// TIA Portal V20 export
// export: Created 2026-04-20T18:50:18.1743947Z, ExportSetting WithDefaults, DisplayName Totally Integrated Automation Portal, DisplayVersion V20, DisplayName TIA Portal Openness, DisplayVersion V20, DisplayName TIA Portal Version Control Interface, DisplayVersion V20, DisplayName STEP 7 Professional, DisplayVersion V20, DisplayName STEP 7 Safety, DisplayVersion V20, DisplayName WinCC Basic/Comfort/Advanced, DisplayVersion V20
TYPE "UDT_AlarmLimits"
// ============================================================
//  BlockParam Demo - Process Plant Structure (Setpoints + Comments)
//  Author: Tobias Laubscher
//  Target: TIA Portal V17+
//  Comment language: en-GB
// 
//  Import procedure:
//    1. Set TIA project editing language to English (United Kingdom)
//    2. Add as external source, then "Generate blocks from source"
//    3. Verify Setpoint flags and comments on a sample member
// 
//  Hierarchy depth from DB root to leaf:
//    DB -> units[] -> modules[] -> valves[] -> *Limits -> hiLimit  (5 levels)
// 
//  Setpoint policy:
//    - Tunable parameters and every parent container on the path
//      carry { S7_SetPoint := 'True' }
//    - Identification / metadata members (tags, names, IDs) do not
//  ============================================================
// stored: IsFailsafeCompliant false
   STRUCT
      hiHiLimit { S7_SetPoint := 'True'} : Real := 100.0;   // Upper critical alarm limit, action required
      hiLimit { S7_SetPoint := 'True'} : Real := 90.0;   // Upper warning alarm limit
      loLimit { S7_SetPoint := 'True'} : Real := 10.0;   // Lower warning alarm limit
      loLoLimit { S7_SetPoint := 'True'} : Real := 5.0;   // Lower critical alarm limit, action required
      hysteresis { S7_SetPoint := 'True'} : Real := 0.5;   // Alarm hysteresis to prevent chattering
      alarmDelay { S7_SetPoint := 'True'} : Time := T#3S;   // Delay before alarm is raised
      enable { S7_SetPoint := 'True'} : Bool := TRUE;   // Enable alarm monitoring for this limit set
   END_STRUCT;
END_TYPE
